PROGRAM LEDs
VAR
	rgbw	:	RGBW;
END_VAR

rgbw();

END_PROGRAM

(* stored: Version 1.1.0.1, ProductVersion 3.1.4024.12
   POU LEDs: Id {080668ae-5330-4f9e-94a4-ce20fb139d33}, SpecialFunc None *)
